TYPE PTOChannelCompact :
STRUCT
	{attribute addProperty Name "PTO Status"}
	PTOStatus : PTOstatusChannel;
	{attribute addProperty Name "ENC Status compact"}
	ENCStatusCompact : ENCStatusCompactChannel;
	{attribute addProperty Name "PTO Control"}
	PTOControl : PTOcontrolChannel;
	{attribute addProperty Name "PTO Target compact"}
	PTOTargetCompact : PTOTargetCompactChannel;
	{attribute addProperty Name "ENC Control compact"}
	ENCControlCompact : ENCControlCompactChannel;
END_STRUCT
END_TYPE

(* stored: Version 1.1.0.1, ProductVersion 3.1.4024.9
   DUT PTOChannelCompact: Id {4f994eca-eb92-08ad-2f00-82da20754acc} *)
